// TIA Portal V18 export
TYPE "PLCtoMES_ST350_ext"
// stored: IsFailsafeCompliant false
   STRUCT
      MainCheckIn { S7_SetPoint := 'True'} : "PLCtoMES_MainCheckIn_ext";   // PLC发送主件请求交互数据到MES
      SubCheckIn { S7_SetPoint := 'True'} : "PLCtoMES_SubCheckIn_ext";
      ScanResultsStored { S7_SetPoint := 'True'} : "PLCtoMES_ResultsStoredScanExchange_ext";   // PLC发送Processing请求,表明工件已经入不可逆工艺,比如压装工位等
      PrintExchange { S7_SetPoint := 'True'} : "PLCtoMES_PrintExchange_ext";   // PLC发送打印交互数据到MES
      MainCheckOut { S7_SetPoint := 'True'} : "PLCtoMES_MainCheckOut_ext";   // PLC发送保存请求到MES
      Common { S7_SetPoint := 'True'} : "PLCtoMES_Common_ext";
   END_STRUCT;
END_TYPE
